{attribute 'qualified_only'}
VAR_GLOBAL
END_VAR

(* stored: Version 1.1.0.1, ProductVersion 3.1.4024.12
   GVL GVL_SP1L0: Id {0162de12-1607-4af5-8d16-e1c7cc4821e0} *)
